# B&R Automation Studio project pneutrunk_plc_experiments
Automation Studio 4.9

## Configuration Config1

### Task classes (Cpu.sw)
```
Cyclic#1:
  Client <- Source.UDP.Client.prg [disabled]
  Narazy <- Source.Narazy.prg [disabled]
  Server <- Source.UDP.Server.prg [disabled]
  Receiver <- (binary)
  Sender <- (binary)
Cyclic#2:
  test_input <- test_input.prg (AdditionalIncludeDirectories=\Logical\MATLAB_includes\R2023a\, BuildOptions=-lm -DMODEL=simulink_2_plc -DNUMST=2 -DNCSTATES=0 -DHAVESTDIO -DRT -DUSE_RTMODEL -DEXT_MODE -DEXTMODE_STATIC -DEXTMODE_STATIC_SIZE=1000000 -DON_TARGET_WAIT_FOR_START=0 -DCLASSIC_INTERFACE=1 -DALLOCATIONFCN=0 -DTID01EQ=1 -DMAT_FILE=0 -DONESTEPFCN=0 -DTERMFCN=1 -DMULTI_INSTANCE_CODE=0 -DINTEGER_CODE=0 -DMT=0 )
Cyclic#3:
  solo_reg <- solo_reg.prg (AdditionalIncludeDirectories=\Logical\MATLAB_includes\R2023a\, BuildOptions=-lm -DMODEL=pneutr2_reg_FF_stiff -DNUMST=1 -DNCSTATES=0 -DHAVESTDIO -DRT -DUSE_RTMODEL -DCLASSIC_INTERFACE=1 -DALLOCATIONFCN=0 -DTID01EQ=0 -DMAT_FILE=0 -DONESTEPFCN=0 -DTERMFCN=1 -DMULTI_INSTANCE_CODE=0 -DINTEGER_CODE=0 -DMT=0 )
Cyclic#4:
  Receiver1 <- Source.RS485.Receiver.prg
  Sender1 <- Source.RS485.Sender.prg
  Identifika <- Source.Identifikacia.prg [disabled]
  meranie <- meranie.prg [disabled] (AdditionalIncludeDirectories=\Logical\MATLAB_includes\R2022b\, BuildOptions=-lm -DMODEL=pneutrunkMeranie -DNUMST=1 -DNCSTATES=0 -DHAVESTDIO -DRT -DUSE_RTMODEL -DEXT_MODE -DEXTMODE_STATIC -DEXTMODE_STATIC_SIZE=1000000 -DON_TARGET_WAIT_FOR_START=0 -DCLASSIC_INTERFACE=1 -DALLOCATIONFCN=0 -DTID01EQ=0 -DMAT_FILE=0 -DONESTEPFCN=0 -DTERMFCN=1 -DMULTI_INSTANCE_CODE=0 -DINTEGER_CODE=0 -DMT=0 )
  Testing <- Source.Testing.prg [disabled]
  Program <- Source.Program.prg [disabled]
  Repeatabil <- Source.Experiments.Repeatability.prg
Cyclic#5:
  Controller <- Source.Controller.prg
DataObjects: Acp10sys
Binaries: FWRules, TCData, udbdef, asfw, User, iomap, sysconf, arconfig, ashwd, Role, ashwac, Acp10map, acp10cfg
Libraries: runtime, AsUDP, asstring, standard, sys_lib, brsystem, dvframe, AsTCP, AsArLog, regulatory, asieccon, astime, powerlnk, fileio
```

## Logical view

### Global.typ - Global data types
```iecst
TYPE
	tlacidla : 	STRUCT
		start : BOOL;
		ros : BOOL;
		stopLED : BOOL;
		stop : BOOL;
		startLED : BOOL;
		startButton : BOOL;
		centralStop : BOOL;
		stropBielaLED : BOOL;
		stropCervenaLED : BOOL;
		klucik : BOOL;
	END_STRUCT;
	automatic : 	STRUCT
		y_desired : ARRAY[0..6]OF INT := [7(0)];
		x_desired : ARRAY[0..6]OF INT := [7(0)];
		linear : INT;
		ball_up : BOOL;
		casovac : BOOL;
		effector : BOOL;
		casovac_uchopenie : BOOL;
		ball_piston : BOOL;
		novyCyklus : TIME := T#1s;
		novyCyklusStart : BOOL;
		trajectoryStart2 : BOOL;
		trajectoryTime2 : TIME := T#6s;
		automatic : BOOL;
		holdPosition : BOOL;
		cas : INT;
		box : INT;
		step_color : INT;
		popcorn : BOOL;
		testFarba : INT;
		loptickyVzasobniku : BOOL := TRUE;
		x_desired_previous : ARRAY[0..6]OF INT;
		y_desired_previous : ARRAY[0..6]OF INT;
		I_konstanta : ARRAY[0..6]OF INT;
		levitacia : BOOL;
		desiredPressure2 : ARRAY[0..6]OF INT;
		desiredPressure3 : ARRAY[0..6]OF INT;
		desiredPressure3_previous : ARRAY[0..6]OF INT;
		desiredPressure2_previous : ARRAY[0..6]OF INT;
		desiredPressure1_previous : ARRAY[0..6]OF INT;
		desiredPressureLinear : INT;
		desiredPressure1 : ARRAY[0..6]OF INT;
		repeatability : BOOL;
	END_STRUCT;
	podavac : 	STRUCT
		levitovanie : BOOL;
		ball_piston_sjf : BOOL;
		ball : BOOL;
		ball_piston : BOOL;
	END_STRUCT;
	identifikacia : 	STRUCT
		p3 : REAL;
		p2 : REAL;
		p1 : REAL;
		vzorka : USINT;
		uhol2 : ARRAY[0..9]OF INT;
		uhol2Priemer : INT;
		uhol1Priemer : INT;
		uhol1 : ARRAY[0..9]OF INT;
		uhol2Stabilny : BOOL;
		uhol1Stabilny : BOOL;
		uhol2Ref : INT;
		uhol1Ref : INT;
		krok : USINT;
		p2Mem : REAL;
		p1Mem : REAL;
		tonStart : BOOL;
		pocetOverenie : USINT := 10;
		spustit : BOOL;
		p3Koniec : BOOL;
		p2Koniec : BOOL;
		p1Koniec : BOOL;
		p3Mem : REAL;
		results : INT;
		switchs : BOOL;
		inkrement : REAL;
		hornyTlak : REAL;
	END_STRUCT;
	packetRS485 : 	STRUCT
		packet : ARRAY[0..9]OF BYTE;
		sendPacketLED : ARRAY[0..5]OF BYTE;
		sendPacketSnimace : ARRAY[0..5]OF BYTE;
		sendPacketFinal : ARRAY[0..5]OF BYTE;
		id : USINT;
	END_STRUCT;
	packetUDP : 	STRUCT
		qLength : INT;
		c : INT;
		q : INT;
		qFull : STRING[80];
		comma : INT;
		qString : ARRAY[0..14]OF STRING[6];
		qDesired : ARRAY[0..14]OF REAL;
		color : INT;
		step : INT;
	END_STRUCT;
	tlaky : 	STRUCT
		tlak3 : USINT;
		tlak2 : USINT;
		tlak1 : USINT;
	END_STRUCT;
	moduly : 	STRUCT
		uhol2 : ARRAY[0..6]OF REAL := [7(0.0)];
		uhol1 : ARRAY[0..6]OF REAL := [7(0.0)];
		koncak : ARRAY[0..6]OF BOOL;
		led : ARRAY[0..6]OF BOOL;
		uholINT2 : INT;
		uholINT1 : INT;
		tlak1 : ARRAY[0..6]OF INT;
		tlak2 : ARRAY[0..6]OF INT;
		tlak3 : ARRAY[0..6]OF INT;
		tlakLinear : INT;
		uhol_XminusRef : ARRAY[0..6]OF REAL; (*uhol ktory posiela PLC do PC po odpocitani odchylky naklonenia realneho robota*)
		uhol_YminusRef : ARRAY[0..6]OF REAL; (*uhol ktory posiela PLC do PC po odpocitani odchylky naklonenia realneho robota*)
		linearReal : REAL;
		naraz : ARRAY[0..7]OF BOOL;
		narazAktivny : BOOL;
	END_STRUCT;
END_TYPE
```

### Global.var - Global variables
```iecst
VAR
	hranica_upravy_traj : REAL := 2;
	Yellow_tab_ID7 : REAL;
	zasobnik : podavac;
	Yellow_tab_ID6 : REAL;
	I_ON : BOOL;
	Yellow_tab_ID5 : REAL;
	step : INT;
	Yellow_tab_ID4 : REAL;
	Yellow_tab_ID3 : REAL;
	Yellow_tab_ID2 : REAL;
	automatika : automatic;
	Yellow_tab_ID1 : REAL;
	u2 : INT;
	u1 : INT;
	stiffness_ff : REAL;
	result : INT;
	RESET_ID7 : REAL;
	RESET_ID6 : REAL;
	RESET_ID5 : REAL;
	RESET_ID4 : REAL;
	RESET_ID3 : REAL;
	RESET_ID2 : REAL;
	RESET_ID1 : REAL;
	ref_linearny_posun : REAL;
	ref_alfa_y_ID7 : REAL;
	ref_alfa_y_ID6 : REAL;
	ref_alfa_y_ID5 : REAL;
	ref_alfa_y_ID4 : REAL;
	ref_alfa_y_ID3 : REAL;
	ref_alfa_y_ID2 : REAL;
	ref_alfa_y_ID1 : REAL;
	ref_alfa_x_ID7 : REAL;
	ref_alfa_x_ID6 : REAL;
	ref_alfa_x_ID5 : REAL;
	ref_alfa_x_ID4 : REAL;
	ref_alfa_x_ID3 : REAL;
	ref_alfa_x_ID2 : REAL;
	ref_alfa_x_ID1 : REAL;
	q_real : ARRAY[0..12] OF REAL := [0.55,12.58,12.23,7.85,1.23,15.36,17.85,12.05,3.85,3.6,-12.52,10.65,31.28];
	q_desired : ARRAY[0..12] OF REAL;
	pripustna_odchylka_naklonenia : REAL := 0.25;
	poradie_ID7 : REAL;
	poradie_ID6 : REAL;
	poradie_ID5 : REAL;
	poradie_ID4 : REAL;
	poradie_ID3 : REAL;
	poradie_ID2 : REAL;
	poradie_ID1 : REAL;
	packetPos : packetUDP;
	packet485 : packetRS485;
	p3 : REAL;
	p2 : REAL;
	p1 : REAL;
	modul : moduly;
	meranie : identifikacia;
	lin_pressure : REAL;
	I_konstanta_ID7 : REAL;
	I_konstanta_ID6 : REAL;
	I_konstanta_ID5 : REAL;
	I_konstanta_ID4 : REAL;
	I_konstanta_ID3 : REAL;
	I_konstanta_ID2 : REAL;
	cos_test_hodnota2 : REAL;
	cos_test_hodnota1 : REAL;
	I_konstanta_ID1 : REAL;
	Green_tab_ID7 : REAL;
	Green_tab_ID6 : REAL;
	trajectoryStart : BOOL;
	Green_tab_ID5 : REAL;
	Green_tab_ID4 : REAL;
	Green_tab_ID3 : REAL;
	Green_tab_ID2 : REAL;
	Green_tab_ID1 : REAL;
	step_color : INT;
	global_step_udp : INT;
	global_step : INT;
	datagramLength : INT;
	centralStop : BOOL;
	cas_trajektorie : REAL := 100;
	Blue_tab_ID7 : REAL;
	Blue_tab_ID6 : REAL;
	Blue_tab_ID5 : REAL;
	buttons : tlacidla;
	Blue_tab_ID4 : REAL;
	Blue_tab_ID3 : REAL;
	Blue_tab_ID2 : REAL;
	Blue_tab_ID1 : REAL;
	act_alfa_y_ID7 : REAL;
	act_alfa_y_ID6 : REAL;
	act_alfa_y_ID5 : REAL;
	step_repeatability : INT;
	act_alfa_y_ID4 : REAL;
	act_alfa_y_ID3 : REAL;
	act_alfa_y_ID2 : REAL;
	act_alfa_y_ID1 : REAL;
	act_alfa_x_ID7 : REAL;
	act_alfa_x_ID6 : REAL;
	act_alfa_x_ID5 : REAL;
	act_alfa_x_ID4 : REAL;
	act_alfa_x_ID3 : REAL;
	act_alfa_x_ID2 : REAL;
	act_alfa_x_ID1 : REAL;
END_VAR
```

### Package Logical/Libraries - Global libraries

### Program Logical/Libraries/regulatory

#### regulatory.typ
```iecst
TYPE
	emxArray_real_T :  STRUCT
		data :  REFERENCE TO LREAL;
		size :  REFERENCE TO DINT;
		allocatedSize :  DINT;
		numDimensions :  DINT;
		canFreeData :  BOOL;
	END_STRUCT;

	B_regulator_FF_PI_T :  STRUCT
		Input1 :  REAL;
		Input2 :  REAL;
		Input3 :  REAL;
		Input4 :  REAL;
		Input11 :  REAL;
		Input5 :  REAL;
		Input13 :  REAL;
		Input14 :  REAL;
		Input8 :  REAL;
		Input9 :  REAL;
		Input10 :  REAL;
		Sum :  REAL;
		Input7 :  REAL;
		Sum2 :  REAL;
		Input6 :  REAL;
		Sum1 :  REAL;
		Input12 :  REAL;
	END_STRUCT;

	DW_regulator_FF_PI_T :  STRUCT
		Integrator_DSTATE :  LREAL;
		Filter_DSTATE :  LREAL;
		Integrator_DSTATE_o :  LREAL;
		Filter_DSTATE_f :  LREAL;
		Integrator_DSTATE_i :  LREAL;
		Filter_DSTATE_a :  LREAL;
		Integrator_PrevResetState :  SINT;
		Filter_PrevResetState :  SINT;
		Integrator_PrevResetState_l :  SINT;
		Filter_PrevResetState_e :  SINT;
		Integrator_PrevResetState_e :  SINT;
		Filter_PrevResetState_h :  SINT;
	END_STRUCT;

	ConstP_regulator_FF_PI_T :  STRUCT
		Constant_Value_m :  ARRAY[0..113] OF REAL;
		Constant1_Value_b :  ARRAY[0..113] OF REAL;
		Constant2_Value :  ARRAY[0..113] OF REAL;
		Constant3_Value :  ARRAY[0..113] OF REAL;
	END_STRUCT;

	tag_RTM_regulator_FF_PI_T :  STRUCT
		errorStatus :  REFERENCE TO USINT;
		blockIO :  REFERENCE TO B_regulator_FF_PI_T;
		dwork :  REFERENCE TO DW_regulator_FF_PI_T;
	END_STRUCT;

	B_regulator_FF_PI_plane_regre_T :  STRUCT
		Input1 :  REAL;
		Input2 :  REAL;
		Input3 :  REAL;
		Input4 :  REAL;
		Input11 :  REAL;
		Input5 :  REAL;
		Input13 :  REAL;
		Input14 :  REAL;
		Sum :  REAL;
		Input7 :  REAL;
		Sum2 :  REAL;
		Input6 :  REAL;
		Sum1 :  REAL;
		Input10 :  REAL;
		Input12 :  REAL;
		Input8 :  REAL;
		Input9 :  REAL;
	END_STRUCT;

	DW_regulator_FF_PI_plane_regr_T :  STRUCT
		Integrator_DSTATE :  LREAL;
		Filter_DSTATE :  LREAL;
		Integrator_DSTATE_o :  LREAL;
		Filter_DSTATE_f :  LREAL;
		Integrator_DSTATE_i :  LREAL;
		Filter_DSTATE_a :  LREAL;
		Integrator_PrevResetState :  SINT;
		Filter_PrevResetState :  SINT;
		Integrator_PrevResetState_l :  SINT;
		Filter_PrevResetState_e :  SINT;
		Integrator_PrevResetState_e :  SINT;
		Filter_PrevResetState_h :  SINT;
	END_STRUCT;

	tag_RTM_regulator_FF_PI_plane_T :  STRUCT
		errorStatus :  REFERENCE TO USINT;
		blockIO :  REFERENCE TO B_regulator_FF_PI_plane_regre_T;
		dwork :  REFERENCE TO DW_regulator_FF_PI_plane_regr_T;
	END_STRUCT;

	B_PID_constant_T :  STRUCT
		Input1 :  REAL;
		Input2 :  REAL;
		Input3 :  REAL;
		Input4 :  REAL;
		Input11 :  REAL;
		Input5 :  REAL;
		Input13 :  REAL;
		Input14 :  REAL;
		Switch2 :  REAL;
		Input6 :  REAL;
		Switch1 :  REAL;
		Input7 :  REAL;
		Switch :  REAL;
		Input12 :  REAL;
	END_STRUCT;

	DW_PID_constant_T :  STRUCT
		Integrator_DSTATE :  LREAL;
		Filter_DSTATE :  LREAL;
		Integrator_DSTATE_f :  LREAL;
		Filter_DSTATE_j :  LREAL;
		Integrator_DSTATE_h :  LREAL;
		Filter_DSTATE_m :  LREAL;
		Integrator_PrevResetState :  SINT;
		Filter_PrevResetState :  SINT;
		Integrator_PrevResetState_m :  SINT;
		Filter_PrevResetState_e :  SINT;
		Integrator_PrevResetState_l :  SINT;
		Filter_PrevResetState_k :  SINT;
	END_STRUCT;

	tag_RTM_PID_constant_T :  STRUCT
		errorStatus :  REFERENCE TO USINT;
		blockIO :  REFERENCE TO B_PID_constant_T;
		dwork :  REFERENCE TO DW_PID_constant_T;
	END_STRUCT;

	B_requestedalfa2deltaz1_reg_F_T :  STRUCT
		Blue_real :  REAL;
		Green_real :  REAL;
		Yellow_real :  REAL;
		Blue_ref :  REAL;
		Green_ref :  REAL;
		Yellow_ref :  REAL;
	END_STRUCT;

	B_regulator_nelin_P_T :  STRUCT
		Input1 :  REAL;
		Input2 :  REAL;
		Input3 :  REAL;
		Input4 :  REAL;
		Gain7 :  REAL;
		Gain9 :  REAL;
		Gain8 :  REAL;
	END_STRUCT;

	tag_RTM_regulator_nelin_P_T :  STRUCT
		errorStatus :  REFERENCE TO USINT;
		blockIO :  REFERENCE TO B_regulator_nelin_P_T;
	END_STRUCT;

	B_PID_co_T :  STRUCT
		Input1 :  REAL;
		Input2 :  REAL;
		Input3 :  REAL;
		Input4 :  REAL;
		Input11 :  REAL;
		Input5 :  REAL;
		Input13 :  REAL;
		Input14 :  REAL;
		Switch2 :  REAL;
		Input6 :  REAL;
		Switch1 :  REAL;
		Input7 :  REAL;
		Switch :  REAL;
		Input12 :  REAL;
	END_STRUCT;

	DW_PID_co_T :  STRUCT
		Integrator_DSTATE :  LREAL;
		Filter_DSTATE :  LREAL;
		Integrator_DSTATE_f :  LREAL;
		Filter_DSTATE_j :  LREAL;
		Integrator_DSTATE_h :  LREAL;
		Filter_DSTATE_m :  LREAL;
		Integrator_PrevResetState :  SINT;
		Filter_PrevResetState :  SINT;
		Integrator_PrevResetState_m :  SINT;
		Filter_PrevResetState_e :  SINT;
		Integrator_PrevResetState_l :  SINT;
		Filter_PrevResetState_k :  SINT;
	END_STRUCT;

	tag_RTM_PID_co_T :  STRUCT
		errorStatus :  REFERENCE TO USINT;
		blockIO :  REFERENCE TO B_PID_co_T;
		dwork :  REFERENCE TO DW_PID_co_T;
	END_STRUCT;

	B_reg_FF_PI_pl_regr_stiff_T :  STRUCT
		Input15 :  REAL;
		Input1 :  REAL;
		Input2 :  REAL;
		Input3 :  REAL;
		Input4 :  REAL;
		Input16 :  REAL;
		Input11 :  REAL;
		Input5 :  REAL;
		Input13 :  REAL;
		Input14 :  REAL;
		Input17 :  REAL;
		Sum :  REAL;
		Input7 :  REAL;
		Sum2 :  REAL;
		Input6 :  REAL;
		Sum1 :  REAL;
		Input10 :  REAL;
		Input12 :  REAL;
		Input8 :  REAL;
		Input9 :  REAL;
	END_STRUCT;

	DW_reg_FF_PI_pl_regr_stiff_T :  STRUCT
		Integrator_DSTATE :  LREAL;
		Filter_DSTATE :  LREAL;
		Integrator_DSTATE_o :  LREAL;
		Filter_DSTATE_f :  LREAL;
		Integrator_DSTATE_i :  LREAL;
		Filter_DSTATE_a :  LREAL;
		Integrator_PrevResetState :  SINT;
		Filter_PrevResetState :  SINT;
		Integrator_PrevResetState_l :  SINT;
		Filter_PrevResetState_e :  SINT;
		Integrator_PrevResetState_e :  SINT;
		Filter_PrevResetState_h :  SINT;
	END_STRUCT;

	ConstP_reg_FF_PI_pl_regr_stif_T :  STRUCT
		Constant_Value :  ARRAY[0..47] OF LREAL;
		Constant1_Value :  ARRAY[0..47] OF LREAL;
		pooled1 :  ARRAY[0..47] OF LREAL;
		Constant13_Value :  ARRAY[0..47] OF LREAL;
		Constant14_Value :  ARRAY[0..47] OF LREAL;
		pooled2 :  ARRAY[0..47] OF LREAL;
		Constant2_Value :  ARRAY[0..47] OF LREAL;
		Constant3_Value :  ARRAY[0..47] OF LREAL;
		Constant4_Value :  ARRAY[0..47] OF LREAL;
		pooled3 :  ARRAY[0..47] OF LREAL;
		Constant8_Value :  ARRAY[0..47] OF LREAL;
		Constant9_Value :  ARRAY[0..47] OF LREAL;
	END_STRUCT;

	tag_RTM_reg_FF_PI_pl_regr_sti_T :  STRUCT
		errorStatus :  REFERENCE TO USINT;
		blockIO :  REFERENCE TO B_reg_FF_PI_pl_regr_stiff_T;
		dwork :  REFERENCE TO DW_reg_FF_PI_pl_regr_stiff_T;
	END_STRUCT;

	emxArray_real_T_regulator_FF_T2 :emxArray_real_T;	(*  *)

	RT_MODEL_regulator_FF_PI_T :tag_RTM_regulator_FF_PI_T;	(*  *)

	RT_MODEL_regulator_FF_PI_plan_T :tag_RTM_regulator_FF_PI_plane_T;	(*  *)

	RT_MODEL_PID_constant_T :tag_RTM_PID_constant_T;	(*  *)

	RT_MODEL_regulator_nelin_P_T :tag_RTM_regulator_nelin_P_T;	(*  *)

	RT_MODEL_PID_co_T :tag_RTM_PID_co_T;	(*  *)

	RT_MODEL_reg_FF_PI_pl_regr_st_T :tag_RTM_reg_FF_PI_pl_regr_sti_T;	(*  *)

END_TYPE
```

#### reg_FF_PI_pl_regr_stiff_types.h
```c
/*
 * reg_FF_PI_pl_regr_stiff_types.h
 *
 * Academic License - for use in teaching, academic research, and meeting
 * course requirements at degree granting institutions only.  Not for
 * government, commercial, or other organizational use.
 *
 * Code generation for model "reg_FF_PI_pl_regr_stiff".
 *
 * Model version              : 1.154
 * Simulink Coder version : 9.6 (R2021b) 14-May-2021
 * C source code generated on : Mon Jun 26 09:10:26 2023
 *
 * Target selection: bur_grt.tlc
 * Note: GRT includes extra infrastructure and instrumentation for prototyping
 * Embedded hardware selection: Intel->x86/Pentium
 * Code generation objectives: Unspecified
 * Validation result: Not run
 */

#ifndef RTW_HEADER_reg_FF_PI_pl_regr_stiff_types_h_
#define RTW_HEADER_reg_FF_PI_pl_regr_stiff_types_h_

/* Model Code Variants */

/* Forward declaration for rtModel */

#endif                         /* RTW_HEADER_reg_FF_PI_pl_regr_stiff_types_h_ */
```

#### regulator_nelin_P_private.h
```c
/*
 * regulator_nelin_P_private.h
 *
 * Academic License - for use in teaching, academic research, and meeting
 * course requirements at degree granting institutions only.  Not for
 * government, commercial, or other organizational use.
 *
 * Code generation for model "regulator_nelin_P".
 *
 * Model version              : 1.10
 * Simulink Coder version : 9.6 (R2021b) 14-May-2021
 * C source code generated on : Fri Jul 29 10:48:17 2022
 *
 * Target selection: bur_grt.tlc
 * Note: GRT includes extra infrastructure and instrumentation for prototyping
 * Embedded hardware selection: Intel->x86/Pentium
 * Code generation objectives: Unspecified
 * Validation result: Not run
 */

#ifndef RTW_HEADER_regulator_nelin_P_private_h_
#define RTW_HEADER_regulator_nelin_P_private_h_
#include "rtwtypes.h"
#include "multiword_types.h"
#if !defined(rt_VALIDATE_MEMORY)
#define rt_VALIDATE_MEMORY(S, ptr)     if(!(ptr)) {\
 rtmSetErrorStatus(regulator_nelin_P_M, RT_MEMORY_ALLOCATION_ERROR);\
 }
#endif

#if !defined(rt_FREE)
#if !defined(_WIN32)
#define rt_FREE(ptr)                   if((ptr) != (NULL)) {\
 free((ptr));\
 (ptr) = (NULL);\
 }
#else

/* Visual and other windows compilers declare free without const */
#define rt_FREE(ptr)                   if((ptr) != (NULL)) {\
 free((void *)(ptr));\
 (ptr) = (NULL);\
 }
#endif
#endif
#endif                             /* RTW_HEADER_regulator_nelin_P_private_h_ */
```

#### rtmodel.h
```c
/*
 *  rtmodel.h:
 *
 * Academic License - for use in teaching, academic research, and meeting
 * course requirements at degree granting institutions only.  Not for
 * government, commercial, or other organizational use.
 *
 * Code generation for model "regulator_FF_PI".
 *
 * Model version              : 1.65
 * Simulink Coder version : 9.6 (R2021b) 14-May-2021
 * C source code generated on : Tue Mar 22 08:25:51 2022
 *
 * Target selection: bur_grt.tlc
 * Note: GRT includes extra infrastructure and instrumentation for prototyping
 * Embedded hardware selection: Intel->x86/Pentium
 * Code generation objectives: Unspecified
 * Validation result: Not run
 */

#ifndef RTW_HEADER_rtmodel_h_
#define RTW_HEADER_rtmodel_h_

/*
 *  Includes the appropriate headers when we are using rtModel
 */
#include "regulator_FF_PI.h"
#include "regulator_FF_PI_plane_regress.h"
#include "reg_FF_PI_pl_regr_stiff.h"
#include "PID_co.h"
#include "regulator_nelin_P.h"
#define GRTINTERFACE                   0

/*
 * ROOT_IO_FORMAT: 0 (Individual arguments)
 * ROOT_IO_FORMAT: 1 (Structure reference)
 * ROOT_IO_FORMAT: 2 (Part of model data structure)
 */
#define ROOT_IO_FORMAT                 2

/* Macros generated for backwards compatibility  */
#ifndef rtmGetStopRequested
#define rtmGetStopRequested(rtm)       ((void*) 0)
#endif
#endif                                 /* RTW_HEADER_rtmodel_h_ */
```

#### PID_c.c
```c
/********************************************************************
 * COPYRIGHT -- B&R Industrial Automation GmbH
 ********************************************************************
 * Program: regulatory
 * File: regulatory.c
 * Author: MartinV
 * Last modified by: MartinV
 * Created: 26-Sep-2022 14:44:03
 * Last modified: Mon Sep 26 14:43:43 2022
 * Model Version: 1.9
 * Description:
 * modified Comment:
 ********************************************************************
 * Implementation of program regulatory
 ********************************************************************
 * Generated with B&R Automation Studio Target for Simulink V6.5
 * (GRT based)
 ********************************************************************/

#include <bur/plctypes.h>

#include "rtwtypes.h"
#include "rtmodel.h"

#define EXPAND_CONCAT(name1,name2) name1 ## name2
#define CONCAT(name1,name2) EXPAND_CONCAT(name1,name2)
#define RT_MODEL            CONCAT(MODEL,_rtModel)

#ifdef __cplusplus

extern "C" {

#endif

/* Defines */
#define SS_TERMINATE 4
#define SS_OUTPUT 3
#define SS_INITIALIZE 2

#ifdef __cplusplus

}

#endif

#ifdef __cplusplus
    unsigned long bur_heap_size = 6553500;
#endif

void PID_c(struct PID_c* inst)
{
  tag_RTM_PID_co_T* const PID_co_M = &(inst)->bur_PID_co;
	inst->bur_PID_co.blockIO = &(inst)->bur_B_PID_co_T;
	inst->bur_PID_co.dwork = &(inst)->bur_DW_PID_co_T;

  switch (inst->ssMethodType)
  {
    case SS_INITIALIZE:

      /* call model initialize functions */
		/*memInit function */
		PID_co_initializeMemory(PID_co_M, inst);
		PID_co_initialize(PID_co_M, inst);
      break;

    case SS_OUTPUT:
      /* call model step functions */
		PID_co_step(PID_co_M, inst);
      break;

    case SS_TERMINATE:
      /* call model terminate function */
		PID_co_terminate(PID_co_M, inst);
	  break;
  }
}

/*****************************************************************************
   Function block sample time: 0.002
 *****************************************************************************/

/*****************************************************************************
   B&R Automation Studio Target for Simulink Version: V6.5.1 (03-Dec-2021)
 *****************************************************************************/
```

### Program Logical/Source/Controller (IEC)

#### Cyclic.st - Cyclic code
```iecst
PROGRAM _CYCLIC

	TON_0(IN := kalibraciaStart, PT := T#5s0ms);

	IF buttons.klucik = FALSE THEN
		global_step		:= 0;
		step 			:= 7;
		buttons.stropBielaLED	:= FALSE;
	END_IF

	CASE step OF

		0:  // Detekcia referencnej polohy
			IF switch2 = FALSE THEN
				buttons.startLED				:= FALSE;
				switch2 						:= TRUE;
				FOR id:=0 TO 6 BY 1 DO
					modul.tlak1[id]	:= REAL_TO_INT(0);
					modul.tlak2[id]	:= REAL_TO_INT(0);
					modul.tlak3[id]	:= REAL_TO_INT(0);
					packetPos.qDesired[id*2] 	:= 0;
					packetPos.qDesired[id*2+1] 	:= 0;
					automatika.x_desired[id]	:= 0;
					automatika.y_desired[id]	:= 0;
					switch						:= FALSE;
				END_FOR

			END_IF

			IF buttons.startButton = TRUE THEN
				buttons.start	:= TRUE;
				global_step_udp	:= 0;
			END_IF

			IF buttons.start = TRUE AND buttons.centralStop = TRUE THEN
				buttons.stop					:= FALSE;
				buttons.stopLED					:= FALSE;
				buttons.stropCervenaLED			:= FALSE;
				buttons.startLED				:= TRUE;
				IF switch = FALSE THEN
					switch 						:= TRUE;
					kalibraciaStart 			:= TRUE;
					I_ON						:= TRUE;
					FOR id:=0 TO 6 BY 1 DO
						automatika.I_konstanta[id]	:= 25;
					END_FOR
					FOR id:=0 TO 6 BY 1 DO
						modul.tlak1[id]			:= REAL_TO_INT(3*32767/9);
						modul.tlak2[id]			:= REAL_TO_INT(3*32767/9);
						modul.tlak3[id]			:= REAL_TO_INT(3*32767/9);
					END_FOR
				END_IF

				IF switch = TRUE AND TON_0.Q = TRUE THEN
					switch			:= FALSE;
					kalibraciaStart	:= FALSE;
					step			:= 1;
				END_IF
			END_IF
			global_step				:= 0;
			buttons.stropBielaLED	:= TRUE;
		1:	// Vypustenie vzduchu zo vsetkych mechov, zapnutie I-regulatora
			(*
			FOR id:=0 TO 6 BY 1 DO
				modul.tlak1[id]	:= 0;
				modul.tlak2[id]	:= 0;
				modul.tlak3[id]	:= 0;
			END_FOR
			*)
			//I_ON					:= TRUE;
			switch2 				:= FALSE;
			kalibraciaStart			:= TRUE;

			step					:= 2;

		2:	// cakaj
			IF TON_0.Q = TRUE THEN
				kalibraciaStart		:= FALSE;
				step				:= 3;
			END_IF

		3:
			FOR id:=0 TO 6 BY 1 DO
				modull.nula_x[id]:= 0;
				modull.nula_y[id]:= 0;
			END_FOR

			step					:= 44;

			global_step 			:= 999;
			global_step_udp			:= 0;			// aby nahodou nemal na zaciatku gesto z predoslej udalosti

			kalibraciaStart			:= TRUE;
			(*
			FOR id:=0 TO 6 BY 1 DO
				modul.tlak1[id]	:= 0;
				modul.tlak2[id]	:= 0;
				modul.tlak3[id]	:= 0;
			END_FOR
			*)

		44:
			IF TON_0.Q = TRUE THEN
				kalibraciaStart		:= FALSE;
				step				:= 4;
				FOR id:=0 TO 6 BY 1 DO
					modull.nula_x[id]:= modul.uhol1[id];
					modull.nula_y[id]:= modul.uhol2[id];
				END_FOR
			END_IF

		4:

			FOR id:=0 TO 6 BY 1 DO
				modull.real_uhol_x_kalibrovane[id]	:= modul.uhol1[id];
				modull.real_uhol_y_kalibrovane[id]	:= modul.uhol2[id];
			//	modul.uhol_XminusRef[id] 			:= modull.real_uhol_x_kalibrovane[id] - modull.nula_x[id];
			//	modul.uhol_YminusRef[id] 			:= modull.real_uhol_y_kalibrovane[id] - modull.nula_y[id];
				modul.linearReal		 			:= ref_linearny_posun;
			END_FOR

			IF (automatika.step_color = 1 OR automatika.step_color = 2) AND global_step = 0 THEN
				global_step			:= 999;
			END_IF

			zasobnik.ball			:= automatika.ball_up;
			zasobnik.ball_piston	:= automatika.ball_piston;
			zasobnik.ball_piston_sjf:= automatika.popcorn;
			zasobnik.levitovanie	:= automatika.levitacia;
			modull.efektor			:= automatika.effector;
			I_konstanta_ID1			:= automatika.I_konstanta[0];
			I_konstanta_ID2			:= automatika.I_konstanta[1];
			I_konstanta_ID3			:= automatika.I_konstanta[2];
			I_konstanta_ID4			:= automatika.I_konstanta[3];
			I_konstanta_ID5			:= automatika.I_konstanta[4];
			I_konstanta_ID6			:= automatika.I_konstanta[5];
			I_konstanta_ID7			:= automatika.I_konstanta[6];

			IF buttons.stop = TRUE THEN
				buttons.start		:= FALSE;
				buttons.startLED	:= FALSE;
				buttons.stopLED		:= TRUE;
				global_step			:= 7;
			END_IF

			IF buttons.start = TRUE AND buttons.centralStop = TRUE THEN
				IF automatika.automatic = TRUE THEN
					IF automatika.holdPosition = FALSE THEN
						FOR id:=0 TO 6 BY 1 DO
							modull.pozadovany_uhol_y[id]	:=  packetPos.qDesired[id*2];
							modull.pozadovany_uhol_x[id]	:= -packetPos.qDesired[id*2+1];
						END_FOR
						modull.pozadovanyLinear				:= packetPos.qDesired[14]*7/25 + 23;
					END_IF
				ELSE
					FOR id:=0 TO 6 BY 1 DO
						modull.pozadovany_uhol_x[id]	:= automatika.x_desired[id];
						modull.pozadovany_uhol_y[id] 	:= automatika.y_desired[id];
					END_FOR
					modull.pozadovanyLinear				:= automatika.linear;
				END_IF

				// Joint limits
				FOR id:=0 TO 6 BY 1 DO
					IF modull.pozadovany_uhol_x[id] >= maxUhol THEN
						modull.pozadovany_uhol_x[id]	:= maxUhol;
					ELSIF modull.pozadovany_uhol_x[id] <= - maxUhol THEN
						modull.pozadovany_uhol_x[id] := -maxUhol;
					END_IF

					IF modull.pozadovany_uhol_y[id] >= maxUhol THEN
						modull.pozadovany_uhol_y[id]	:= maxUhol;
					ELSIF modull.pozadovany_uhol_y[id] <= - maxUhol THEN
						modull.pozadovany_uhol_y[id] := -maxUhol;
					END_IF

				END_FOR

				ref_alfa_x_ID1:= modull.pozadovany_uhol_x[0];
				ref_alfa_y_ID1:= modull.pozadovany_uhol_y[0];
				ref_alfa_x_ID2:= modull.pozadovany_uhol_x[1];
				ref_alfa_y_ID2:= modull.pozadovany_uhol_y[1];
				ref_alfa_x_ID3:= modull.pozadovany_uhol_x[2];
				ref_alfa_y_ID3:= modull.pozadovany_uhol_y[2];
				ref_alfa_x_ID4:= modull.pozadovany_uhol_x[3];
				ref_alfa_y_ID4:= modull.pozadovany_uhol_y[3];
				ref_alfa_x_ID5:= modull.pozadovany_uhol_x[4];
				ref_alfa_y_ID5:= modull.pozadovany_uhol_y[4];
				ref_alfa_x_ID6:= modull.pozadovany_uhol_x[5];
				ref_alfa_y_ID6:= modull.pozadovany_uhol_y[5];
				ref_alfa_x_ID7:= modull.pozadovany_uhol_x[6];
				ref_alfa_y_ID7:= modull.pozadovany_uhol_y[6];

				// Obmedzenie pre linearny posun (ak je hodnota nad 30 regulator sa sprava divne, nechce sa vypnut)
				IF modull.pozadovanyLinear >30 THEN
					ref_linearny_posun	:= 30;
				ELSIF modull.pozadovanyLinear <23 THEN
					ref_linearny_posun	:= 23;
				ELSE
					ref_linearny_posun	:= modull.pozadovanyLinear;
				END_IF

				act_alfa_x_ID1:= modull.real_uhol_x_kalibrovane[0] - modull.nula_x[0];
				act_alfa_y_ID1:= modull.real_uhol_y_kalibrovane[0] - modull.nula_y[0];
				act_alfa_x_ID2:= modull.real_uhol_x_kalibrovane[1] - modull.nula_x[1];
				act_alfa_y_ID2:= modull.real_uhol_y_kalibrovane[1] - modull.nula_y[1];
				act_alfa_x_ID3:= modull.real_uhol_x_kalibrovane[2] - modull.nula_x[2];
				act_alfa_y_ID3:= modull.real_uhol_y_kalibrovane[2] - modull.nula_y[2];
				act_alfa_x_ID4:= modull.real_uhol_x_kalibrovane[3] - modull.nula_x[3];
				act_alfa_y_ID4:= modull.real_uhol_y_kalibrovane[3] - modull.nula_y[3];
				act_alfa_x_ID5:= modull.real_uhol_x_kalibrovane[4] - modull.nula_x[4];
				act_alfa_y_ID5:= modull.real_uhol_y_kalibrovane[4] - modull.nula_y[4];
				act_alfa_x_ID6:= modull.real_uhol_x_kalibrovane[5] - modull.nula_x[5];
				act_alfa_y_ID6:= modull.real_uhol_y_kalibrovane[5] - modull.nula_y[5];
				act_alfa_x_ID7:= modull.real_uhol_x_kalibrovane[6] - modull.nula_x[6];
				act_alfa_y_ID7:= modull.real_uhol_y_kalibrovane[6] - modull.nula_y[6];

				IF automatika.repeatability = FALSE THEN

					// Nastavenie tlakov podla regulacie
					// ID1
					id:=0;
					modul.tlak1[id] := REAL_TO_INT(Blue_tab_ID1*32767/9);
					modul.tlak2[id] := REAL_TO_INT(Green_tab_ID1*32767/9);
					modul.tlak3[id] := REAL_TO_INT(Yellow_tab_ID1*32767/9);

					// ID2
					id:=1;
					modul.tlak1[id] := REAL_TO_INT(Blue_tab_ID2*32767/9);
					modul.tlak2[id] := REAL_TO_INT(Green_tab_ID2*32767/9);
					modul.tlak3[id] := REAL_TO_INT(Yellow_tab_ID2*32767/9);

					// ID3
					id:=2;
					modul.tlak1[id] := REAL_TO_INT(Blue_tab_ID3*32767/9);
					modul.tlak2[id] := REAL_TO_INT(Green_tab_ID3*32767/9);
					modul.tlak3[id] := REAL_TO_INT(Yellow_tab_ID3*32767/9);

					// ID4
					id:=3;
					modul.tlak1[id] := REAL_TO_INT(Blue_tab_ID4*32767/9);
					modul.tlak2[id] := REAL_TO_INT(Green_tab_ID4*32767/9);
					modul.tlak3[id] := REAL_TO_INT(Yellow_tab_ID4*32767/9);

					// ID5
					id:=4;
					modul.tlak1[id] := REAL_TO_INT(Blue_tab_ID5*32767/9);
					modul.tlak2[id] := REAL_TO_INT(Green_tab_ID5*32767/9);
					modul.tlak3[id] := REAL_TO_INT(Yellow_tab_ID5*32767/9);

					// ID6
					id:=5;
					modul.tlak1[id] := REAL_TO_INT(Blue_tab_ID6*32767/9);
					modul.tlak2[id] := REAL_TO_INT(Green_tab_ID6*32767/9);
					modul.tlak3[id] := REAL_TO_INT(Yellow_tab_ID6*32767/9);

					// ID7
					id:=6;
					modul.tlak3[id] := REAL_TO_INT(Blue_tab_ID7*32767/9);
					modul.tlak1[id] := REAL_TO_INT(Green_tab_ID7*32767/9);
					modul.tlak2[id] := REAL_TO_INT(Yellow_tab_ID7*32767/9);

					//lin_modul
					modul.tlakLinear:= REAL_TO_INT(lin_pressure*32767/9);
				ELSE
					FOR id:= 0 TO 5 BY 1 DO
						modul.tlak1[id] := automatika.desiredPressure1[id];
						modul.tlak2[id] := automatika.desiredPressure2[id];
						modul.tlak3[id] := automatika.desiredPressure3[id];
					END_FOR
					modul.tlakLinear	:= automatika.desiredPressureLinear;
				END_IF

			ELSIF buttons.centralStop = FALSE OR buttons.start = FALSE THEN
				buttons.start			:= FALSE;
				switch					:= FALSE;
				switch2					:= FALSE;
				I_ON					:= FALSE;
				kalibraciaStart			:= FALSE;
				step					:= 0;
				global_step_udp			:= 0;
				global_step				:= 0;
				step_repeatability		:= 0;
				automatika.repeatability:= FALSE;
				automatika.casovac		:= FALSE;
				automatika.ball_piston	:= FALSE;
				automatika.ball_up		:= FALSE;
				automatika.levitacia	:= FALSE;
				zasobnik.levitovanie	:= FALSE;
				zasobnik.ball_piston_sjf:= FALSE;
				automatika.popcorn		:= FALSE;
				automatika.casovac_uchopenie:= FALSE;
				automatika.effector		:= FALSE;
				automatika.holdPosition	:= FALSE;
				automatika.automatic	:= FALSE;
				act_alfa_x_ID1:= 0;
				act_alfa_y_ID1:= 0;
				act_alfa_x_ID2:= 0;
				act_alfa_y_ID2:= 0;
				act_alfa_x_ID3:= 0;
				act_alfa_y_ID3:= 0;
				act_alfa_x_ID4:= 0;
				act_alfa_y_ID4:= 0;
				act_alfa_x_ID5:= 0;
				act_alfa_y_ID5:= 0;
				act_alfa_x_ID6:= 0;
				act_alfa_y_ID6:= 0;
				act_alfa_x_ID7:= 0;
				act_alfa_y_ID7:= 0;
				ref_alfa_x_ID1:= 0;
				ref_alfa_y_ID1:= 0;
				ref_alfa_x_ID2:= 0;
				ref_alfa_y_ID2:= 0;
				ref_alfa_x_ID3:= 0;
				ref_alfa_y_ID3:= 0;
				ref_alfa_x_ID4:= 0;
				ref_alfa_y_ID4:= 0;
				ref_alfa_x_ID5:= 0;
				ref_alfa_y_ID5:= 0;
				ref_alfa_x_ID6:= 0;
				ref_alfa_y_ID6:= 0;
				ref_alfa_x_ID7:= 0;
				ref_alfa_y_ID7:= 0;
				FOR i:=0 TO 6 BY 1 DO
					modul.tlak1[i] 				:= 0;
					modul.tlak2[i]				:= 0;
					modul.tlak3[i] 				:= 0;
					modull.pozadovany_uhol_y[i]	:= 0;
					modull.pozadovany_uhol_x[i]	:= 0;
					modull.real_uhol_x_kalibrovane[i]	:= 0;
					modull.real_uhol_y_kalibrovane[i] 	:= 0;
					modull.nula_x[i]			:= 0;
					modull.nula_y[i]			:= 0;
				END_FOR
				modul.tlakLinear		:= 0;
				modull.efektor			:= FALSE;
				modull.pozadovanyLinear	:= 23;
				zasobnik.ball			:= FALSE;
				zasobnik.ball_piston	:= FALSE;
			END_IF
		5: // kolaborativny mod - doslo k narazu, alebo stlacenie stop
			buttons.startLED			:= FALSE;
			buttons.stopLED				:= TRUE;
			IF buttons.start = TRUE THEN
				buttons.stropBielaLED	:= FALSE;
				buttons.stropCervenaLED	:= TRUE;
				buttons.start			:= FALSE;
			END_IF
			step						:= 6;
			global_step					:= 0;

		6:
			IF buttons.stop = TRUE THEN
				buttons.stopLED			:= FALSE;
				buttons.stropCervenaLED	:= FALSE;
				buttons.stropBielaLED	:= TRUE;
				step					:= 7;
			END_IF

		7:	// resetovanie vsetkeho
			buttons.start			:= FALSE;
			switch					:= FALSE;
			switch2					:= FALSE;
			I_ON					:= FALSE;
			kalibraciaStart			:= FALSE;
			step					:= 0;
			global_step_udp			:= 0;
			global_step				:= 0;
			automatika.casovac		:= FALSE;
			zasobnik.levitovanie	:= FALSE;
			zasobnik.ball_piston_sjf:= FALSE;
			automatika.ball_piston	:= FALSE;
			automatika.ball_up		:= FALSE;
			automatika.popcorn		:= FALSE;
			zasobnik.ball_piston_sjf:= FALSE;
			automatika.casovac_uchopenie:= FALSE;
			automatika.effector		:= FALSE;
			automatika.holdPosition	:= FALSE;
			automatika.automatic	:= FALSE;
			act_alfa_x_ID1:= 0;
			act_alfa_y_ID1:= 0;
			act_alfa_x_ID2:= 0;
			act_alfa_y_ID2:= 0;
			act_alfa_x_ID3:= 0;
			act_alfa_y_ID3:= 0;
			act_alfa_x_ID4:= 0;
			act_alfa_y_ID4:= 0;
			act_alfa_x_ID5:= 0;
			act_alfa_y_ID5:= 0;
			act_alfa_x_ID6:= 0;
			act_alfa_y_ID6:= 0;
			act_alfa_x_ID7:= 0;
			act_alfa_y_ID7:= 0;
			ref_alfa_x_ID1:= 0;
			ref_alfa_y_ID1:= 0;
			ref_alfa_x_ID2:= 0;
			ref_alfa_y_ID2:= 0;
			ref_alfa_x_ID3:= 0;
			ref_alfa_y_ID3:= 0;
			ref_alfa_x_ID4:= 0;
			ref_alfa_y_ID4:= 0;
			ref_alfa_x_ID5:= 0;
			ref_alfa_y_ID5:= 0;
			ref_alfa_x_ID6:= 0;
			ref_alfa_y_ID6:= 0;
			ref_alfa_x_ID7:= 0;
			ref_alfa_y_ID7:= 0;
			FOR i:=0 TO 6 BY 1 DO
				modul.tlak1[i] 				:= 0;
				modul.tlak2[i]				:= 0;
				modul.tlak3[i] 				:= 0;
				modull.pozadovany_uhol_y[i]	:= 0;
				modull.pozadovany_uhol_x[i]	:= 0;
				modull.real_uhol_x_kalibrovane[i]	:= 0;
				modull.real_uhol_y_kalibrovane[i] 	:= 0;
				modull.nula_x[i]			:= 0;
				modull.nula_y[i]			:= 0;
			END_FOR
			modul.tlakLinear		:= 0;
			modull.efektor			:= FALSE;
			modull.pozadovanyLinear	:= 23;
			zasobnik.ball			:= FALSE;
			zasobnik.ball_piston	:= FALSE;
			IF buttons.klucik = FALSE THEN
				step				:= 8;
				global_step			:= 0;
			ELSE
				step				:= 0;
			END_IF
		8:
			IF buttons.klucik = TRUE THEN
				step				:= 0;
				global_step			:= 0;
			ELSE
				buttons.stropBielaLED	:= FALSE;
			END_IF

	END_CASE

	IF I_ON= TRUE THEN
		RESET_ID1:= TRUE;
		RESET_ID2:= TRUE;
		RESET_ID3:= TRUE;
		RESET_ID4:= TRUE;
		RESET_ID5:= TRUE;
		RESET_ID6:= TRUE;
		RESET_ID7:= TRUE;
	ELSE
		RESET_ID1:= FALSE;
		RESET_ID2:= FALSE;
		RESET_ID3:= FALSE;
		RESET_ID4:= FALSE;
		RESET_ID5:= FALSE;
		RESET_ID6:= FALSE;
		RESET_ID7:= FALSE;
	END_IF

	I_konstanta_ID1;
	I_konstanta_ID2;
	I_konstanta_ID3;
	I_konstanta_ID4;
	I_konstanta_ID5;
	I_konstanta_ID6;
	I_konstanta_ID7;

END_PROGRAM
```

#### Variables.var - Local variables
```iecst
VAR
	Vin_x_prechodne : REAL;
	Vin_y_prechodne : REAL;
	pocitadlo : INT;
	Vin_x_priemer : REAL;
	Vin_y_priemer : REAL;
	cos_test : BOOL;
	kalibracia_x : REAL;
	kalibracia_y : REAL;
	uhol_y_predosly : REAL;
	uhol_x_predosly : REAL;
	pozadovany_uhol_y_predosly : REAL;
	x1 : REAL := 5;
	y1 : REAL := 75;
	x2 : REAL := 1;
	y2 : REAL := 350;
	a : REAL;
	b : REAL;
	error_x : REAL;
	error_total : REAL;
	error_y : REAL;
	modull : mech;
	test_const_I : BOOL := FALSE;
	pozadovany_uhol_x_predosly : REAL;
	p11 : REAL;
	p22 : REAL;
	p33 : REAL;
	stlacene : BOOL;
	poradie : INT;
	pozadovany_uhol_x_old : REAL;
	pozadovany_uhol_y_old : REAL;
	i : INT;
	FF_PID_r_t_3 : FF_PID_r_t;
	FF_PID_r_t_0 : FF_PID_r_t;
	id : INT;
	FF_PID_r_t_1 : FF_PID_r_t;
	FF_PID_r_t_2 : FF_PID_r_t;
	switch : BOOL;
	maxUhol : INT;
	TON_0 : TON;
	kalibraciaStart : BOOL;
	TON_1 : TON;
	switch2 : BOOL;
END_VAR
```

### Program Logical/Source/Identifikacia (IEC)

#### Variables.var
```iecst
VAR
	cMod : INT;
	i : INT;
	TON_0 : TON;
	TON_1 : TON;
END_VAR
```

### Program Logical/Source/Experiments/Repeatability (IEC)

#### Variables.var
```iecst
VAR
	casovac_start : BOOL;
	step_repeatability : USINT;
	TON_0 : TON;
	i : INT;
	TON_1 : TON;
	pauza : BOOL;
END_VAR
```

#### Cyclic.st
```iecst
PROGRAM _CYCLIC

	TON_0(IN := casovac_start, PT := INT_TO_TIME(automatika.cas));
	TON_1(IN := pauza, PT := T#3s0ms);

	IF step = 4 THEN

		CASE step_repeatability OF
			0:
				casovac_start				:= TRUE;
				step_repeatability			:= 1;
				automatika.repeatability	:= TRUE;
				automatika.cas				:= 5000;

			1:	// Point A
				automatika.desiredPressure1[0]:= TIME_TO_INT(TON_0.ET)*1669/((automatika.cas));
				automatika.desiredPressure1[1]:= TIME_TO_INT(TON_0.ET)*3013/((automatika.cas));
				automatika.desiredPressure1[2]:= TIME_TO_INT(TON_0.ET)*(-4146)/((automatika.cas));
				automatika.desiredPressure1[3]:= TIME_TO_INT(TON_0.ET)*(-8424)/((automatika.cas));
				automatika.desiredPressure1[4]:= TIME_TO_INT(TON_0.ET)*335/((automatika.cas));
				automatika.desiredPressure1[5]:= TIME_TO_INT(TON_0.ET)*2453/((automatika.cas));
				automatika.desiredPressure1[6]:= TIME_TO_INT(TON_0.ET)*6053/((automatika.cas));

				automatika.desiredPressure2[0]:= TIME_TO_INT(TON_0.ET)*6958/((automatika.cas));
				automatika.desiredPressure2[1]:= TIME_TO_INT(TON_0.ET)*4381/((automatika.cas));
				automatika.desiredPressure2[2]:= TIME_TO_INT(TON_0.ET)*12008/((automatika.cas));
				automatika.desiredPressure2[3]:= TIME_TO_INT(TON_0.ET)*13312/((automatika.cas));
				automatika.desiredPressure2[4]:= TIME_TO_INT(TON_0.ET)*8361/((automatika.cas));
				automatika.desiredPressure2[5]:= TIME_TO_INT(TON_0.ET)*6761/((automatika.cas));
				automatika.desiredPressure2[6]:= TIME_TO_INT(TON_0.ET)*3567/((automatika.cas));

				automatika.desiredPressure3[0]:= TIME_TO_INT(TON_0.ET)*4006/((automatika.cas));
				automatika.desiredPressure3[1]:= TIME_TO_INT(TON_0.ET)*5379/((automatika.cas));
				automatika.desiredPressure3[2]:= TIME_TO_INT(TON_0.ET)*5605/((automatika.cas));
				automatika.desiredPressure3[3]:= TIME_TO_INT(TON_0.ET)*3560/((automatika.cas));
				automatika.desiredPressure3[4]:= TIME_TO_INT(TON_0.ET)*3900/((automatika.cas));
				automatika.desiredPressure3[5]:= TIME_TO_INT(TON_0.ET)*3205/((automatika.cas));
				automatika.desiredPressure3[6]:= TIME_TO_INT(TON_0.ET)*2770/((automatika.cas));

				automatika.desiredPressureLinear := TIME_TO_INT(TON_0.ET)*10800/((automatika.cas));

				IF TON_0.Q = TRUE THEN
					casovac_start		:= FALSE;
					step_repeatability	:= 2;
					FOR i:=0 TO 6 BY 1 DO
						automatika.desiredPressure1_previous[i]		:= automatika.desiredPressure1[i];
						automatika.desiredPressure2_previous[i]		:= automatika.desiredPressure2[i];
						automatika.desiredPressure3_previous[i]		:= automatika.desiredPressure3[i];
					END_FOR
				END_IF

			2:	// Pause
				pauza					:= TRUE;
				step_repeatability		:= 3;
			3:
				IF TON_1.Q = TRUE THEN
					pauza				:= FALSE;
					step_repeatability	:= 4;
					casovac_start		:= TRUE;
				END_IF

			4:	// Point B
				automatika.desiredPressure1[0]:= (automatika.desiredPressure1_previous[0]*(automatika.cas - TIME_TO_INT(TON_0.ET))/automatika.cas) + TIME_TO_INT(TON_0.ET)*(5403)/(automatika.cas);
				automatika.desiredPressure1[1]:= (automatika.desiredPressure1_previous[1]*(automatika.cas - TIME_TO_INT(TON_0.ET))/automatika.cas) + TIME_TO_INT(TON_0.ET)*(5622)/(automatika.cas);
				automatika.desiredPressure1[2]:= (automatika.desiredPressure1_previous[2]*(automatika.cas - TIME_TO_INT(TON_0.ET))/automatika.cas) + TIME_TO_INT(TON_0.ET)*(7940)/(automatika.cas);
				automatika.desiredPressure1[3]:= (automatika.desiredPressure1_previous[3]*(automatika.cas - TIME_TO_INT(TON_0.ET))/automatika.cas) + TIME_TO_INT(TON_0.ET)*(6420)/(automatika.cas);
				automatika.desiredPressure1[4]:= (automatika.desiredPressure1_previous[4]*(automatika.cas - TIME_TO_INT(TON_0.ET))/automatika.cas) + TIME_TO_INT(TON_0.ET)*(8355)/(automatika.cas);
				automatika.desiredPressure1[5]:= (automatika.desiredPressure1_previous[5]*(automatika.cas - TIME_TO_INT(TON_0.ET))/automatika.cas) + TIME_TO_INT(TON_0.ET)*(6516)/(automatika.cas);
				automatika.desiredPressure1[6]:= (automatika.desiredPressure1_previous[6]*(automatika.cas - TIME_TO_INT(TON_0.ET))/automatika.cas) + TIME_TO_INT(TON_0.ET)*(565)/(automatika.cas);

				automatika.desiredPressure2[0]:= (automatika.desiredPressure2_previous[0]*(automatika.cas - TIME_TO_INT(TON_0.ET))/automatika.cas) + TIME_TO_INT(TON_0.ET)*(1406)/(automatika.cas);
				automatika.desiredPressure2[1]:= (automatika.desiredPressure2_previous[1]*(automatika.cas - TIME_TO_INT(TON_0.ET))/automatika.cas) + TIME_TO_INT(TON_0.ET)*(2287)/(automatika.cas);
				automatika.desiredPressure2[2]:= (automatika.desiredPressure2_previous[2]*(automatika.cas - TIME_TO_INT(TON_0.ET))/automatika.cas) + TIME_TO_INT(TON_0.ET)*(271)/(automatika.cas);
				automatika.desiredPressure2[3]:= (automatika.desiredPressure2_previous[3]*(automatika.cas - TIME_TO_INT(TON_0.ET))/automatika.cas) + TIME_TO_INT(TON_0.ET)*(2520)/(automatika.cas);
				automatika.desiredPressure2[4]:= (automatika.desiredPressure2_previous[4]*(automatika.cas - TIME_TO_INT(TON_0.ET))/automatika.cas) + TIME_TO_INT(TON_0.ET)*(829)/(automatika.cas);
				automatika.desiredPressure2[5]:= (automatika.desiredPressure2_previous[5]*(automatika.cas - TIME_TO_INT(TON_0.ET))/automatika.cas) + TIME_TO_INT(TON_0.ET)*(1928)/(automatika.cas);
				automatika.desiredPressure2[6]:= (automatika.desiredPressure2_previous[6]*(automatika.cas - TIME_TO_INT(TON_0.ET))/automatika.cas) + TIME_TO_INT(TON_0.ET)*(4860)/(automatika.cas);

				automatika.desiredPressure3[0]:= (automatika.desiredPressure3_previous[0]*(automatika.cas - TIME_TO_INT(TON_0.ET))/automatika.cas) + TIME_TO_INT(TON_0.ET)*(5933)/(automatika.cas);
				automatika.desiredPressure3[1]:= (automatika.desiredPressure3_previous[1]*(automatika.cas - TIME_TO_INT(TON_0.ET))/automatika.cas) + TIME_TO_INT(TON_0.ET)*(4731)/(automatika.cas);
				automatika.desiredPressure3[2]:= (automatika.desiredPressure3_previous[2]*(automatika.cas - TIME_TO_INT(TON_0.ET))/automatika.cas) + TIME_TO_INT(TON_0.ET)*(4820)/(automatika.cas);
				automatika.desiredPressure3[3]:= (automatika.desiredPressure3_previous[3]*(automatika.cas - TIME_TO_INT(TON_0.ET))/automatika.cas) + TIME_TO_INT(TON_0.ET)*(3573)/(automatika.cas);
				automatika.desiredPressure3[4]:= (automatika.desiredPressure3_previous[4]*(automatika.cas - TIME_TO_INT(TON_0.ET))/automatika.cas) + TIME_TO_INT(TON_0.ET)*(3796)/(automatika.cas);
				automatika.desiredPressure3[5]:= (automatika.desiredPressure3_previous[5]*(automatika.cas - TIME_TO_INT(TON_0.ET))/automatika.cas) + TIME_TO_INT(TON_0.ET)*(4104)/(automatika.cas);
				automatika.desiredPressure3[6]:= (automatika.desiredPressure3_previous[6]*(automatika.cas - TIME_TO_INT(TON_0.ET))/automatika.cas) + TIME_TO_INT(TON_0.ET)*(7462)/(automatika.cas);

				automatika.desiredPressureLinear := TIME_TO_INT(TON_0.ET)*10800/((automatika.cas));

				IF TON_0.Q = TRUE THEN
					casovac_start		:= FALSE;
					step_repeatability	:= 5;
					FOR i:=0 TO 6 BY 1 DO
						automatika.desiredPressure1_previous[i]	:= automatika.desiredPressure1[i];
						automatika.desiredPressure2_previous[i]	:= automatika.desiredPressure2[i];
						automatika.desiredPressure3_previous[i]	:= automatika.desiredPressure3[i];
					END_FOR
				END_IF
			5:	// Pause
				pauza					:= TRUE;
				step_repeatability		:= 6;
			6:
				IF TON_1.Q = TRUE THEN
					pauza				:= FALSE;
					step_repeatability	:= 7;
					casovac_start		:= TRUE;
				END_IF

			7:	// Point A
				automatika.desiredPressure1[0]:= (automatika.desiredPressure1_previous[0]*(automatika.cas - TIME_TO_INT(TON_0.ET))/automatika.cas) + TIME_TO_INT(TON_0.ET)*(1669)/(automatika.cas);
				automatika.desiredPressure1[1]:= (automatika.desiredPressure1_previous[1]*(automatika.cas - TIME_TO_INT(TON_0.ET))/automatika.cas) + TIME_TO_INT(TON_0.ET)*(3013)/(automatika.cas);
				automatika.desiredPressure1[2]:= (automatika.desiredPressure1_previous[2]*(automatika.cas - TIME_TO_INT(TON_0.ET))/automatika.cas) + TIME_TO_INT(TON_0.ET)*(-4146)/(automatika.cas);
				automatika.desiredPressure1[3]:= (automatika.desiredPressure1_previous[3]*(automatika.cas - TIME_TO_INT(TON_0.ET))/automatika.cas) + TIME_TO_INT(TON_0.ET)*(-8424)/(automatika.cas);
				automatika.desiredPressure1[4]:= (automatika.desiredPressure1_previous[4]*(automatika.cas - TIME_TO_INT(TON_0.ET))/automatika.cas) + TIME_TO_INT(TON_0.ET)*(335)/(automatika.cas);
				automatika.desiredPressure1[5]:= (automatika.desiredPressure1_previous[5]*(automatika.cas - TIME_TO_INT(TON_0.ET))/automatika.cas) + TIME_TO_INT(TON_0.ET)*(2453)/(automatika.cas);
				automatika.desiredPressure1[6]:= (automatika.desiredPressure1_previous[6]*(automatika.cas - TIME_TO_INT(TON_0.ET))/automatika.cas) + TIME_TO_INT(TON_0.ET)*(6053)/(automatika.cas);

				automatika.desiredPressure2[0]:= (automatika.desiredPressure2_previous[0]*(automatika.cas - TIME_TO_INT(TON_0.ET))/automatika.cas) + TIME_TO_INT(TON_0.ET)*(6958)/(automatika.cas);
				automatika.desiredPressure2[1]:= (automatika.desiredPressure2_previous[1]*(automatika.cas - TIME_TO_INT(TON_0.ET))/automatika.cas) + TIME_TO_INT(TON_0.ET)*(4381)/(automatika.cas);
				automatika.desiredPressure2[2]:= (automatika.desiredPressure2_previous[2]*(automatika.cas - TIME_TO_INT(TON_0.ET))/automatika.cas) + TIME_TO_INT(TON_0.ET)*(12008)/(automatika.cas);
				automatika.desiredPressure2[3]:= (automatika.desiredPressure2_previous[3]*(automatika.cas - TIME_TO_INT(TON_0.ET))/automatika.cas) + TIME_TO_INT(TON_0.ET)*(13312)/(automatika.cas);
				automatika.desiredPressure2[4]:= (automatika.desiredPressure2_previous[4]*(automatika.cas - TIME_TO_INT(TON_0.ET))/automatika.cas) + TIME_TO_INT(TON_0.ET)*(8361)/(automatika.cas);
				automatika.desiredPressure2[5]:= (automatika.desiredPressure2_previous[5]*(automatika.cas - TIME_TO_INT(TON_0.ET))/automatika.cas) + TIME_TO_INT(TON_0.ET)*(6761)/(automatika.cas);
				automatika.desiredPressure2[6]:= (automatika.desiredPressure2_previous[6]*(automatika.cas - TIME_TO_INT(TON_0.ET))/automatika.cas) + TIME_TO_INT(TON_0.ET)*(3567)/(automatika.cas);

				automatika.desiredPressure3[0]:= (automatika.desiredPressure3_previous[0]*(automatika.cas - TIME_TO_INT(TON_0.ET))/automatika.cas) + TIME_TO_INT(TON_0.ET)*(4006)/(automatika.cas);
				automatika.desiredPressure3[1]:= (automatika.desiredPressure3_previous[1]*(automatika.cas - TIME_TO_INT(TON_0.ET))/automatika.cas) + TIME_TO_INT(TON_0.ET)*(5379)/(automatika.cas);
				automatika.desiredPressure3[2]:= (automatika.desiredPressure3_previous[2]*(automatika.cas - TIME_TO_INT(TON_0.ET))/automatika.cas) + TIME_TO_INT(TON_0.ET)*(5605)/(automatika.cas);
				automatika.desiredPressure3[3]:= (automatika.desiredPressure3_previous[3]*(automatika.cas - TIME_TO_INT(TON_0.ET))/automatika.cas) + TIME_TO_INT(TON_0.ET)*(3560)/(automatika.cas);
				automatika.desiredPressure3[4]:= (automatika.desiredPressure3_previous[4]*(automatika.cas - TIME_TO_INT(TON_0.ET))/automatika.cas) + TIME_TO_INT(TON_0.ET)*(3900)/(automatika.cas);
				automatika.desiredPressure3[5]:= (automatika.desiredPressure3_previous[5]*(automatika.cas - TIME_TO_INT(TON_0.ET))/automatika.cas) + TIME_TO_INT(TON_0.ET)*(3205)/(automatika.cas);
				automatika.desiredPressure3[6]:= (automatika.desiredPressure3_previous[6]*(automatika.cas - TIME_TO_INT(TON_0.ET))/automatika.cas) + TIME_TO_INT(TON_0.ET)*(2770)/(automatika.cas);

				automatika.desiredPressureLinear := TIME_TO_INT(TON_0.ET)*10800/((automatika.cas));

				IF TON_0.Q = TRUE THEN
					casovac_start		:= FALSE;
					step_repeatability	:= 8;
					FOR i:=0 TO 6 BY 1 DO
						automatika.desiredPressure1_previous[i]	:= automatika.desiredPressure1[i];
						automatika.desiredPressure2_previous[i]	:= automatika.desiredPressure2[i];
						automatika.desiredPressure3_previous[i]	:= automatika.desiredPressure3[i];
					END_FOR
				END_IF
			8:	// Pause
				pauza					:= TRUE;
				step_repeatability		:= 9;
			9:
				IF TON_1.Q = TRUE THEN
					pauza				:= FALSE;
					step_repeatability	:= 4;
					casovac_start		:= TRUE;
				END_IF

		END_CASE

	END_IF

END_PROGRAM
```

### Program Logical/Source/Experiments/Continuum

#### Types.typ
```iecst
TYPE
	tlak : 	STRUCT
		p2 : REAL;
		p3 : REAL;
		p1 : REAL;
	END_STRUCT;
END_TYPE
```

#### Cyclic.st
```iecst
PROGRAM _CYCLIC
	automatika.experiment2	:= TRUE;
	FOR id:=0 TO 5 BY 1 DO
		modul.tlak1[id]	:= REAL_TO_INT(pressure.p1*32767/9);
		modul.tlak2[id]	:= REAL_TO_INT(pressure.p2*32767/9);
		modul.tlak3[id]	:= REAL_TO_INT(pressure.p3*32767/9);
	END_FOR
	(*
	modul.tlak2[6]	:= REAL_TO_INT(pressure.p3*32767/9);
	modul.tlak3[6]	:= REAL_TO_INT(pressure.p2*32767/9);
	modul.tlak1[6]	:= REAL_TO_INT(pressure.p1*32767/9);
	*)
	modul.tlak2[6]	:= REAL_TO_INT(pressure.p3*32767/9);
	modul.tlak3[6]	:= REAL_TO_INT(pressure.p1*32767/9);
	modul.tlak1[6]	:= REAL_TO_INT(pressure.p2*32767/9);
END_PROGRAM
```

### Program Logical/Source/Experiments/HandControl

#### Variables.var
```iecst
VAR
	id : INT;
END_VAR
```

#### Cyclic.st
```iecst
PROGRAM _CYCLIC
	IF automatika.handControl = TRUE THEN
		FOR id:=0 TO 6 BY 1 DO
			automatika.x_desired[id]	:= (uhly.ref_alfa_x[id]);
			automatika.y_desired[id]	:= (uhly.ref_alfa_y[id]);
		END_FOR
	ELSIF automatika.handControl = FALSE THEN
		FOR id:=0 TO 6 BY 1 DO
			automatika.x_desired[id]	:= 0;
			automatika.y_desired[id]	:= 0;
		END_FOR
	END_IF

END_PROGRAM
```

#### Init.st
```iecst
PROGRAM _INIT

	FOR id:=0 TO 6 BY 1 DO
		automatika.I_konstanta[id]	:= 5;
	END_FOR

END_PROGRAM
```

### Program Logical/meranie (ANSIC)

#### pneutrunkMeranie_types.h
```c
/*
 * pneutrunkMeranie_types.h
 *
 * Academic License - for use in teaching, academic research, and meeting
 * course requirements at degree granting institutions only.  Not for
 * government, commercial, or other organizational use.
 *
 * Code generation for model "pneutrunkMeranie".
 *
 * Model version              : 1.6
 * Simulink Coder version : 9.8 (R2022b) 13-May-2022
 * C source code generated on : Wed May 24 11:04:27 2023
 *
 * Target selection: bur_grt.tlc
 * Note: GRT includes extra infrastructure and instrumentation for prototyping
 * Embedded hardware selection: Intel->x86/Pentium
 * Code generation objectives: Unspecified
 * Validation result: Not run
 */

#ifndef RTW_HEADER_pneutrunkMeranie_types_h_
#define RTW_HEADER_pneutrunkMeranie_types_h_

/* Forward declaration for rtModel */
typedef struct tag_RTM_pneutrunkMeranie_T RT_MODEL_pneutrunkMeranie_T;

#endif                                /* RTW_HEADER_pneutrunkMeranie_types_h_ */
```

#### rt_defines.h
```c
/*
 * rt_defines.h
 *
 * Academic License - for use in teaching, academic research, and meeting
 * course requirements at degree granting institutions only.  Not for
 * government, commercial, or other organizational use.
 *
 * Code generation for model "pneutrunkMeranie".
 *
 * Model version              : 1.6
 * Simulink Coder version : 9.8 (R2022b) 13-May-2022
 * C source code generated on : Wed May 24 11:04:27 2023
 *
 * Target selection: bur_grt.tlc
 * Note: GRT includes extra infrastructure and instrumentation for prototyping
 * Embedded hardware selection: Intel->x86/Pentium
 * Code generation objectives: Unspecified
 * Validation result: Not run
 */

#ifndef RTW_HEADER_rt_defines_h_
#define RTW_HEADER_rt_defines_h_

/*===========*
 * Constants *
 *===========*/
#define RT_PI                          3.14159265358979323846
#define RT_PIF                         3.1415927F
#define RT_LN_10                       2.30258509299404568402
#define RT_LN_10F                      2.3025851F
#define RT_LOG10E                      0.43429448190325182765
#define RT_LOG10EF                     0.43429449F
#define RT_E                           2.7182818284590452354
#define RT_EF                          2.7182817F

/*
 * UNUSED_PARAMETER(x)
 *   Used to specify that a function parameter (argument) is required but not
 *   accessed by the function body.
 */
#ifndef UNUSED_PARAMETER
#if defined(__LCC__)
#define UNUSED_PARAMETER(x)                                      /* do nothing */
#else

/*
 * This is the semi-ANSI standard way of indicating that an
 * unused function parameter is required.
 */
#define UNUSED_PARAMETER(x)            (void) (x)
#endif
#endif
#endif                                 /* RTW_HEADER_rt_defines_h_ */
```

#### rt_nonfinite.h
```c
/*
 * rt_nonfinite.h
 *
 * Academic License - for use in teaching, academic research, and meeting
 * course requirements at degree granting institutions only.  Not for
 * government, commercial, or other organizational use.
 *
 * Code generation for model "pneutrunkMeranie".
 *
 * Model version              : 1.6
 * Simulink Coder version : 9.8 (R2022b) 13-May-2022
 * C source code generated on : Wed May 24 11:04:27 2023
 *
 * Target selection: bur_grt.tlc
 * Note: GRT includes extra infrastructure and instrumentation for prototyping
 * Embedded hardware selection: Intel->x86/Pentium
 * Code generation objectives: Unspecified
 * Validation result: Not run
 */

#ifndef RTW_HEADER_rt_nonfinite_h_
#define RTW_HEADER_rt_nonfinite_h_
#include <stddef.h>
#include "rtwtypes.h"
#define NOT_USING_NONFINITE_LITERALS   1

extern real_T rtInf;
extern real_T rtMinusInf;
extern real_T rtNaN;
extern real32_T rtInfF;
extern real32_T rtMinusInfF;
extern real32_T rtNaNF;
extern void rt_InitInfAndNaN(size_t realSize);
extern boolean_T rtIsInf(real_T value);
extern boolean_T rtIsInfF(real32_T value);
extern boolean_T rtIsNaN(real_T value);
extern boolean_T rtIsNaNF(real32_T value);
typedef struct {
  struct {
    uint32_T wordH;
    uint32_T wordL;
  } words;
} BigEndianIEEEDouble;

typedef struct {
  struct {
    uint32_T wordL;
    uint32_T wordH;
  } words;
} LittleEndianIEEEDouble;

typedef struct {
  union {
    real32_T wordLreal;
    uint32_T wordLuint;
  } wordL;
} IEEESingle;

#endif                                 /* RTW_HEADER_rt_nonfinite_h_ */
```

#### rtGetInf.c
```c
/*
 * rtGetInf.c
 *
 * Academic License - for use in teaching, academic research, and meeting
 * course requirements at degree granting institutions only.  Not for
 * government, commercial, or other organizational use.
 *
 * Code generation for model "pneutrunkMeranie".
 *
 * Model version              : 1.6
 * Simulink Coder version : 9.8 (R2022b) 13-May-2022
 * C source code generated on : Wed May 24 11:04:27 2023
 *
 * Target selection: bur_grt.tlc
 * Note: GRT includes extra infrastructure and instrumentation for prototyping
 * Embedded hardware selection: Intel->x86/Pentium
 * Code generation objectives: Unspecified
 * Validation result: Not run
 */

#include "rtwtypes.h"
#include "rtGetInf.h"
#include <stddef.h>
#include "rt_nonfinite.h"
#define NumBitsPerChar                 8U

/*
 * Initialize rtInf needed by the generated code.
 * Inf is initialized as non-signaling. Assumes IEEE.
 */
real_T rtGetInf(void)
{
  size_t bitsPerReal = sizeof(real_T) * (NumBitsPerChar);
  real_T inf = 0.0;
  if (bitsPerReal == 32U) {
    inf = rtGetInfF();
  } else {
    uint16_T one = 1U;
    enum {
      LittleEndian,
      BigEndian
    } machByteOrder = (*((uint8_T *) &one) == 1U) ? LittleEndian : BigEndian;
    switch (machByteOrder) {
     case LittleEndian:
      {
        union {
          LittleEndianIEEEDouble bitVal;
          real_T fltVal;
        } tmpVal;

        tmpVal.bitVal.words.wordH = 0x7FF00000U;
        tmpVal.bitVal.words.wordL = 0x00000000U;
        inf = tmpVal.fltVal;
        break;
      }

     case BigEndian:
      {
        union {
          BigEndianIEEEDouble bitVal;
          real_T fltVal;
        } tmpVal;

        tmpVal.bitVal.words.wordH = 0x7FF00000U;
        tmpVal.bitVal.words.wordL = 0x00000000U;
        inf = tmpVal.fltVal;
        break;
      }
    }
  }

  return inf;
}

/*
 * Initialize rtInfF needed by the generated code.
 * Inf is initialized as non-signaling. Assumes IEEE.
 */
real32_T rtGetInfF(void)
{
  IEEESingle infF;
  infF.wordL.wordLuint = 0x7F800000U;
  return infF.wordL.wordLreal;
}

/*
 * Initialize rtMinusInf needed by the generated code.
 * Inf is initialized as non-signaling. Assumes IEEE.
 */
real_T rtGetMinusInf(void)
{
  size_t bitsPerReal = sizeof(real_T) * (NumBitsPerChar);
  real_T minf = 0.0;
  if (bitsPerReal == 32U) {
    minf = rtGetMinusInfF();
  } else {
    uint16_T one = 1U;
    enum {
      LittleEndian,
      BigEndian
    } machByteOrder = (*((uint8_T *) &one) == 1U) ? LittleEndian : BigEndian;
    switch (machByteOrder) {
     case LittleEndian:
      {
        union {
          LittleEndianIEEEDouble bitVal;
          real_T fltVal;
        } tmpVal;

        tmpVal.bitVal.words.wordH = 0xFFF00000U;
        tmpVal.bitVal.words.wordL = 0x00000000U;
        minf = tmpVal.fltVal;
        break;
      }

     case BigEndian:
      {
        union {
          BigEndianIEEEDouble bitVal;
          real_T fltVal;
        } tmpVal;

        tmpVal.bitVal.words.wordH = 0xFFF00000U;
        tmpVal.bitVal.words.wordL = 0x00000000U;
        minf = tmpVal.fltVal;
        break;
      }
    }
  }

  return minf;
}

/*
 * Initialize rtMinusInfF needed by the generated code.
 * Inf is initialized as non-signaling. Assumes IEEE.
 */
real32_T rtGetMinusInfF(void)
{
  IEEESingle minfF;
  minfF.wordL.wordLuint = 0xFF800000U;
  return minfF.wordL.wordLreal;
}
```

### Program Logical/solo_reg (ANSIC, version 1.00.0)

#### global.txt
```
VAR
	    stiffness_ff : REAL := 0; (*tuhos&#x165; ff regulatora (sum tlakov)*)
	    ref_alfa_x_ID1 : REAL := 0; (*requested alfa x in deg*)
	    ref_alfa_y_ID1 : REAL := 0; (*requested alfa y in deg*)
	    act_alfa_x_ID1 : REAL := 0; (*actual alfa x in deg*)
	    act_alfa_y_ID1 : REAL := 0; (*actual alfa y in deg*)
	    poradie_ID1 : REAL := 0; (*zmena poradia vlnovcou*)
	    pripustna_odchylka_naklonenia : REAL := 0; (*pri celkovej odchylke pod, sa bude brat error=0*)
	    RESET_ID1 : REAL := 0; (*reset regulatora*)
	    cas_trajektorie : REAL := 0; (*spomalenie hodnota*cas_cyklu*)
	    hranica_upravy_traj : REAL := 0; (*ak je zmena uhla pod tuto uroven traj sa neupravuje*)
	    Blue_tab_ID1 : REAL := 0; (*Blue_pressure*)
	    ref_alfa_x_ID4 : REAL := 0; (*requested alfa x in deg*)
	    ref_alfa_y_ID4 : REAL := 0; (*requested alfa y in deg*)
	    act_alfa_x_ID4 : REAL := 0; (*actual alfa x in deg*)
	    act_alfa_y_ID4 : REAL := 0; (*actual alfa y in deg*)
	    poradie_ID4 : REAL := 0; (*zmena poradia vlnovcou*)
	    RESET_ID4 : REAL := 0; (*reset regulatora*)
	    Blue_tab_ID4 : REAL := 0; (*Blue_pressure*)
	    Yellow_tab_ID4 : REAL := 0; (*Yellow_pressure*)
	    ref_alfa_x_ID5 : REAL := 0; (*requested alfa x in deg*)
	    ref_alfa_y_ID5 : REAL := 0; (*requested alfa y in deg*)
	    act_alfa_x_ID5 : REAL := 0; (*actual alfa x in deg*)
	    act_alfa_y_ID5 : REAL := 0; (*actual alfa y in deg*)
	    poradie_ID5 : REAL := 0; (*zmena poradia vlnovcou*)
	    RESET_ID5 : REAL := 0; (*reset regulatora*)
	    Blue_tab_ID5 : REAL := 0; (*Blue_pressure*)
	    Green_tab_ID4 : REAL := 0; (*Green_pressure*)
	    Yellow_tab_ID5 : REAL := 0; (*Yellow_pressure*)
	    Green_tab_ID5 : REAL := 0; (*Green_pressure*)
	    ref_alfa_x_ID6 : REAL := 0; (*requested alfa x in deg*)
	    ref_alfa_y_ID6 : REAL := 0; (*requested alfa y in deg*)
	    act_alfa_x_ID6 : REAL := 0; (*actual alfa x in deg*)
	    act_alfa_y_ID6 : REAL := 0; (*actual alfa y in deg*)
	    poradie_ID6 : REAL := 0; (*zmena poradia vlnovcou*)
	    RESET_ID6 : REAL := 0; (*reset regulatora*)
	    Blue_tab_ID6 : REAL := 0; (*Blue_pressure*)
	    Yellow_tab_ID6 : REAL := 0; (*Yellow_pressure*)
	    Green_tab_ID6 : REAL := 0; (*Green_pressure*)
	    Yellow_tab_ID1 : REAL := 0; (*Yellow_pressure*)
	    ref_alfa_x_ID7 : REAL := 0; (*requested alfa x in deg*)
	    ref_alfa_y_ID7 : REAL := 0; (*requested alfa y in deg*)
	    act_alfa_x_ID7 : REAL := 0; (*actual alfa x in deg*)
	    act_alfa_y_ID7 : REAL := 0; (*actual alfa y in deg*)
	    poradie_ID7 : REAL := 0; (*zmena poradia vlnovcou*)
	    RESET_ID7 : REAL := 0; (*reset regulatora*)
	    Blue_tab_ID7 : REAL := 0; (*Blue_pressure*)
	    Yellow_tab_ID7 : REAL := 0; (*Yellow_pressure*)
	    Green_tab_ID7 : REAL := 0; (*Green_pressure*)
	    ref_alfa_x_ID2 : REAL := 0; (*requested alfa x in deg*)
	    ref_alfa_y_ID2 : REAL := 0; (*requested alfa y in deg*)
	    act_alfa_x_ID2 : REAL := 0; (*actual alfa x in deg*)
	    act_alfa_y_ID2 : REAL := 0; (*actual alfa y in deg*)
	    poradie_ID2 : REAL := 0; (*zmena poradia vlnovcou*)
	    RESET_ID2 : REAL := 0; (*reset regulatora*)
	    Blue_tab_ID2 : REAL := 0; (*Blue_pressure*)
	    Green_tab_ID1 : REAL := 0; (*Green_pressure*)
	    Yellow_tab_ID2 : REAL := 0; (*Yellow_pressure*)
	    Green_tab_ID2 : REAL := 0; (*Green_pressure*)
	    ref_alfa_x_ID3 : REAL := 0; (*requested alfa x in deg*)
	    ref_alfa_y_ID3 : REAL := 0; (*requested alfa y in deg*)
	    act_alfa_x_ID3 : REAL := 0; (*actual alfa x in deg*)
	    act_alfa_y_ID3 : REAL := 0; (*actual alfa y in deg*)
	    poradie_ID3 : REAL := 0; (*zmena poradia vlnovcou*)
	    RESET_ID3 : REAL := 0; (*reset regulatora*)
	    Blue_tab_ID3 : REAL := 0; (*Blue_pressure*)
	    Yellow_tab_ID3 : REAL := 0; (*Yellow_pressure*)
	    Green_tab_ID3 : REAL := 0; (*Green_pressure*)
	    I_konstanta_ID1 : REAL := 0; (*I_zosilnenie*)
	    I_konstanta_ID2 : REAL := 0; (*I_zosilnenie*)
	    I_konstanta_ID3 : REAL := 0; (*I_zosilnenie*)
	    I_konstanta_ID4 : REAL := 0; (*I_zosilnenie*)
	    I_konstanta_ID5 : REAL := 0; (*I_zosilnenie*)
	    I_konstanta_ID6 : REAL := 0; (*I_zosilnenie*)
	    I_konstanta_ID7 : REAL := 0; (*I_zosilnenie*)
	    ref_linearny_posun : REAL := 0; (*linearny modul [mm]*)
	    lin_pressure : REAL := 0; (*lin_motion_pressure*)
END_VAR
```

#### rtGetInf.h
```c
/*
 * rtGetInf.h
 *
 * Academic License - for use in teaching, academic research, and meeting
 * course requirements at degree granting institutions only.  Not for
 * government, commercial, or other organizational use.
 *
 * Code generation for model "pneutr2_reg_FF_stiff".
 *
 * Model version              : 4.30
 * Simulink Coder version : 9.9 (R2023a) 19-Nov-2022
 * C source code generated on : Thu Feb 15 10:44:02 2024
 *
 * Target selection: bur_grt.tlc
 * Note: GRT includes extra infrastructure and instrumentation for prototyping
 * Embedded hardware selection: Intel->x86/Pentium
 * Code generation objectives: Unspecified
 * Validation result: Not run
 */

#ifndef RTW_HEADER_rtGetInf_h_
#define RTW_HEADER_rtGetInf_h_
#include "rt_nonfinite.h"
#include "rtwtypes.h"

extern real_T rtGetInf(void);
extern real32_T rtGetInfF(void);
extern real_T rtGetMinusInf(void);
extern real32_T rtGetMinusInfF(void);

#endif                                 /* RTW_HEADER_rtGetInf_h_ */
```

#### task_properties.txt
```
For manual assignment to hardware configuration please
add the following additional include directories:

\Logical\MATLAB_includes\R2023a\

And the following additional build options:

-lm -DMODEL=pneutr2_reg_FF_stiff -DNUMST=1 -DNCSTATES=0 -DHAVESTDIO -DRT -DUSE_RTMODEL -DCLASSIC_INTERFACE=1 -DALLOCATIONFCN=0 -DTID01EQ=0 -DMAT_FILE=0 -DONESTEPFCN=0 -DTERMFCN=1 -DMULTI_INSTANCE_CODE=0 -DINTEGER_CODE=0 -DMT=0
```

### Program Logical/test_input (ANSIC)

#### rtGetNaN.h
```c
/*
 * rtGetNaN.h
 *
 * Academic License - for use in teaching, academic research, and meeting
 * course requirements at degree granting institutions only.  Not for
 * government, commercial, or other organizational use.
 *
 * Code generation for model "simulink_2_plc".
 *
 * Model version              : 1.4
 * Simulink Coder version : 9.9 (R2023a) 19-Nov-2022
 * C source code generated on : Tue Feb  6 09:08:04 2024
 *
 * Target selection: bur_grt.tlc
 * Note: GRT includes extra infrastructure and instrumentation for prototyping
 * Embedded hardware selection: Intel->x86/Pentium
 * Code generation objectives: Unspecified
 * Validation result: Not run
 */

#ifndef RTW_HEADER_rtGetNaN_h_
#define RTW_HEADER_rtGetNaN_h_
#include "rt_nonfinite.h"
#include "rtwtypes.h"

extern real_T rtGetNaN(void);
extern real32_T rtGetNaNF(void);

#endif                                 /* RTW_HEADER_rtGetNaN_h_ */
```

#### simulink_2_plc_dt.h
```c
/*
 * simulink_2_plc_dt.h
 *
 * Academic License - for use in teaching, academic research, and meeting
 * course requirements at degree granting institutions only.  Not for
 * government, commercial, or other organizational use.
 *
 * Code generation for model "simulink_2_plc".
 *
 * Model version              : 1.4
 * Simulink Coder version : 9.9 (R2023a) 19-Nov-2022
 * C source code generated on : Tue Feb  6 09:08:04 2024
 *
 * Target selection: bur_grt.tlc
 * Note: GRT includes extra infrastructure and instrumentation for prototyping
 * Embedded hardware selection: Intel->x86/Pentium
 * Code generation objectives: Unspecified
 * Validation result: Not run
 */

#include "ext_types.h"

/* data type size table */
static uint_T rtDataTypeSizes[] = {
  sizeof(real_T),
  sizeof(real32_T),
  sizeof(int8_T),
  sizeof(uint8_T),
  sizeof(int16_T),
  sizeof(uint16_T),
  sizeof(int32_T),
  sizeof(uint32_T),
  sizeof(boolean_T),
  sizeof(fcn_call_T),
  sizeof(int_T),
  sizeof(pointer_T),
  sizeof(action_T),
  2*sizeof(uint32_T),
  sizeof(int32_T),
  sizeof(uint_T),
  sizeof(char_T),
  sizeof(uchar_T),
  sizeof(time_T)
};

/* data type name table */
static const char_T * rtDataTypeNames[] = {
  "real_T",
  "real32_T",
  "int8_T",
  "uint8_T",
  "int16_T",
  "uint16_T",
  "int32_T",
  "uint32_T",
  "boolean_T",
  "fcn_call_T",
  "int_T",
  "pointer_T",
  "action_T",
  "timer_uint32_pair_T",
  "physical_connection",
  "uint_T",
  "char_T",
  "uchar_T",
  "time_T"
};

/* data type transitions for block I/O structure */
static DataTypeTransition rtBTransitions[] = {
  { (char_T *)(&simulink_2_plc_B.SineWave), 0, 0, 2 },

  { (char_T *)(&simulink_2_plc_B.Gain), 1, 0, 2 }
};

/* data type transition table for block I/O structure */
static DataTypeTransitionTable rtBTransTable = {
  2U,
  rtBTransitions
};

/* data type transitions for Parameters structure */
static DataTypeTransition rtPTransitions[] = {
  { (char_T *)(&simulink_2_plc_P.SineWave_Amp), 0, 0, 8 },

  { (char_T *)(&simulink_2_plc_P.Gain_Gain), 1, 0, 2 }
};

/* data type transition table for Parameters structure */
static DataTypeTransitionTable rtPTransTable = {
  2U,
  rtPTransitions
};

/* [EOF] simulink_2_plc_dt.h */
```

#### rt_nonfinite.c
```c
/*
 * rt_nonfinite.c
 *
 * Academic License - for use in teaching, academic research, and meeting
 * course requirements at degree granting institutions only.  Not for
 * government, commercial, or other organizational use.
 *
 * Code generation for model "simulink_2_plc".
 *
 * Model version              : 1.4
 * Simulink Coder version : 9.9 (R2023a) 19-Nov-2022
 * C source code generated on : Tue Feb  6 09:08:04 2024
 *
 * Target selection: bur_grt.tlc
 * Note: GRT includes extra infrastructure and instrumentation for prototyping
 * Embedded hardware selection: Intel->x86/Pentium
 * Code generation objectives: Unspecified
 * Validation result: Not run
 */

#include "rtGetNaN.h"
#include "rtGetInf.h"
#include <stddef.h>
#include "rtwtypes.h"
#include "rt_nonfinite.h"
#define NumBitsPerChar                 8U

real_T rtInf;
real_T rtMinusInf;
real_T rtNaN;
real32_T rtInfF;
real32_T rtMinusInfF;
real32_T rtNaNF;

/*
 * Initialize the rtInf, rtMinusInf, and rtNaN needed by the
 * generated code. NaN is initialized as non-signaling. Assumes IEEE.
 */
void rt_InitInfAndNaN(size_t realSize)
{
  (void) (realSize);
  rtNaN = rtGetNaN();
  rtNaNF = rtGetNaNF();
  rtInf = rtGetInf();
  rtInfF = rtGetInfF();
  rtMinusInf = rtGetMinusInf();
  rtMinusInfF = rtGetMinusInfF();
}

/* Test if value is infinite */
boolean_T rtIsInf(real_T value)
{
  return (boolean_T)((value==rtInf || value==rtMinusInf) ? 1U : 0U);
}

/* Test if single-precision value is infinite */
boolean_T rtIsInfF(real32_T value)
{
  return (boolean_T)(((value)==rtInfF || (value)==rtMinusInfF) ? 1U : 0U);
}

/* Test if value is not a number */
boolean_T rtIsNaN(real_T value)
{
  boolean_T result = (boolean_T) 0;
  size_t bitsPerReal = sizeof(real_T) * (NumBitsPerChar);
  if (bitsPerReal == 32U) {
    result = rtIsNaNF((real32_T)value);
  } else {
    union {
      LittleEndianIEEEDouble bitVal;
      real_T fltVal;
    } tmpVal;

    tmpVal.fltVal = value;
    result = (boolean_T)((tmpVal.bitVal.words.wordH & 0x7FF00000) == 0x7FF00000 &&
                         ( (tmpVal.bitVal.words.wordH & 0x000FFFFF) != 0 ||
                          (tmpVal.bitVal.words.wordL != 0) ));
  }

  return result;
}

/* Test if single-precision value is not a number */
boolean_T rtIsNaNF(real32_T value)
{
  IEEESingle tmp;
  tmp.wordL.wordLreal = value;
  return (boolean_T)( (tmp.wordL.wordLuint & 0x7F800000) == 0x7F800000 &&
                     (tmp.wordL.wordLuint & 0x007FFFFF) != 0 );
}
```

#### task_properties.txt
```
For manual assignment to hardware configuration please
add the following additional include directories:

\Logical\MATLAB_includes\R2023a\

And the following additional build options:

-lm -DMODEL=simulink_2_plc -DNUMST=2 -DNCSTATES=0 -DHAVESTDIO -DRT -DUSE_RTMODEL -DEXT_MODE -DEXTMODE_STATIC -DEXTMODE_STATIC_SIZE=1000000 -DON_TARGET_WAIT_FOR_START=0 -DCLASSIC_INTERFACE=1 -DALLOCATIONFCN=0 -DTID01EQ=1 -DMAT_FILE=0 -DONESTEPFCN=0 -DTERMFCN=1 -DMULTI_INSTANCE_CODE=0 -DINTEGER_CODE=0 -DMT=0
```

Listed in the project but not available here: Logical/Source/Program, Logical/Source/UDP, Logical/Source/MATLAB_includes, Logical/Source/riadenie.var, Logical/Source/Controller/Init.st, Logical/Source/Controller/Types.typ, Logical/Source/Controller/Exit.st, Logical/Source/RS485, Logical/Source/Testing, Logical/Source/Narazy, Logical/MATLAB_includes, Logical/solo_reg/local.typ, Logical/solo_reg/local.var, Logical/solo_reg/multiword_types.h, Logical/solo_reg/pneutr2_reg_FF_stiff.c, Logical/solo_reg/pneutr2_reg_FF_stiff.h, Logical/solo_reg/pneutr2_reg_FF_stiff_data.c, Logical/solo_reg/pneutr2_reg_FF_stiff_private.h, Logical/solo_reg/pneutr2_reg_FF_stiff_types.h, Logical/solo_reg/rtGetInf.c, Logical/solo_reg/rtGetNaN.c, Logical/solo_reg/rtGetNaN.h, Logical/solo_reg/rt_defines.h, Logical/solo_reg/rt_nonfinite.c, Logical/solo_reg/rt_nonfinite.h, Logical/solo_reg/rtmodel.h, Logical/solo_reg/rtwtypes.h, Logical/solo_reg/solo_reg.c, Logical/solo_reg/zero_crossing_types.h
